{attribute 'linkalways'} 
{attribute 'no_explicit_call' := 'This FB is a CLASS and must be accessed using methods or properties'}
{attribute 'enable_dynamic_creation'}
FUNCTION_BLOCK Node_ContainerType_Vector_String_SINT EXTENDS Node
VAR
    out : _GUID;
END_VAR

METHOD PUBLIC  Clone : I_Node
VAR
	pNode : POINTER TO Node_ContainerType_Vector_String_SINT;
END_VAR
pNode := __NEW(Node_ContainerType_Vector_String_SINT);
Clone := pNode^;
END_METHOD

METHOD FB_init : BOOL
VAR_INPUT
	bInitRetains : BOOL; // if TRUE, the retain variables are initialized (warm start / cold start)
	bInCopyCode : BOOL;  // if TRUE, the instance afterwards gets moved into the copy code (online change)
END_VAR
AddOutput('out', out);
END_METHOD

METHOD PROTECTED OnExecute
out.Value := ContainerType_Vector_String_SINT;
END_METHOD

END_FUNCTION_BLOCK

(* stored: Version 1.1.0.1, ProductVersion 3.1.4026.17
   POU Node_ContainerType_Vector_String_SINT: Id {710939a4-06cd-00b4-12f3-d1fe7fe723d3}, SpecialFunc None
   Folder Constructor: Id {1f49427b-a429-07c5-1798-6b24f6bed35b}
   Method Clone: Id {4ec10133-6b42-0c7d-210a-d258d8a843d5}
   Method FB_init: Id {1461cdde-bf9d-073c-11c0-100804dfc9dd}
   Method OnExecute: Id {63560655-5cc9-04ad-24c0-0c4a6d6898a7} *)
